(* IEC 61131-3 sources: programs/VI-54/VI-54_20171205/VI-54_20171205/Stations/PLC_VI54/VI-54_171014/Class/SafetyClass, 1 file *)

(* ---- SafetyClass.st ---- *)
(*!
<Class
	Name               = "SafetyClass"
	Revision           = "0.0"
	RealtimeTask       = "false"
	CyclicTask         = "false"
	BackgroundTask     = "false"
	Sigmatek           = "false"
	OSInterface        = "false"
	HighPriority       = "false"
	Automatic          = "false"
	UpdateMode         = "Prescan"
	SharedCommandTable = "true"
	Objectsize         = "(390,300)">
	<Channels>
		<Server Name="SafetyOut1" Visualized="false" Initialize="false" WriteProtected="true" Retentive="false"/>
		<Server Name="SafetyOut2" Visualized="false" Initialize="false" WriteProtected="true" Retentive="false"/>
		<Server Name="SafetyOut3" Visualized="false" Initialize="false" WriteProtected="true" Retentive="false"/>
		<Server Name="SafetyOut4" Visualized="false" Initialize="false" WriteProtected="true" Retentive="false"/>
		<Client Name="CleaningMode" Required="true" Internal="false"/>
		<Client Name="MasterOverrule" Required="true" Internal="false"/>
		<Client Name="SafetyInp1" Required="false" Internal="false"/>
		<Client Name="SafetyInp2" Required="false" Internal="false"/>
		<Client Name="SafetyInp3" Required="false" Internal="false"/>
		<Client Name="SafetyInp4" Required="false" Internal="false"/>
	</Channels>
</Class>
*)
SafetyClass : CLASS
  //Servers:
	SafetyOut1 	: SvrChCmd_DINT;
	SafetyOut2 	: SvrCh_DINT;
	SafetyOut3 	: SvrCh_DINT;
	SafetyOut4 	: SvrCh_DINT;
  //Clients:
	MasterOverrule 	: CltCh_DINT;
	CleaningMode 	: CltCh_DINT;
	SafetyInp1 	: CltCh_DINT;
	SafetyInp2 	: CltCh_DINT;
	SafetyInp3 	: CltCh_DINT;
	SafetyInp4 	: CltCh_DINT;
  //Variables:
  //Functions:

	FUNCTION VIRTUAL GLOBAL SafetyOut1::Read
		VAR_OUTPUT
			output (EAX) 	: DINT;
		END_VAR;

	FUNCTION VIRTUAL GLOBAL SafetyOut2::Read
		VAR_OUTPUT
			output (EAX) 	: DINT;
		END_VAR;

	FUNCTION VIRTUAL GLOBAL SafetyOut3::Read
		VAR_OUTPUT
			output (EAX) 	: DINT;
		END_VAR;

	FUNCTION VIRTUAL GLOBAL SafetyOut4::Read
		VAR_OUTPUT
			output (EAX) 	: DINT;
		END_VAR;
  //Tables:
	FUNCTION @STD
		VAR_OUTPUT
			ret_code	: CONFSTATES;
		END_VAR;
	FUNCTION GLOBAL TAB @CT_;
END_CLASS;

FUNCTION VIRTUAL GLOBAL SafetyClass::SafetyOut1::Read
	VAR_OUTPUT
		output (EAX) 	: DINT;
	END_VAR

  SafetyInp1 := SafetyInp1.Read();
  if MasterOverrule.Read() = 1 | CleaningMode.Read() = 1 then
	  SafetyOut1 := 1;
  else
    SafetyOut1 := SafetyInp1;
  end_if;
  SafetyOut1.Write(input:= SafetyOut1);
  Output := SafetyOut1;

END_FUNCTION

FUNCTION VIRTUAL GLOBAL SafetyClass::SafetyOut2::Read
	VAR_OUTPUT
		output (EAX) 	: DINT;
	END_VAR

  SafetyInp2 := SafetyInp2.Read();
  if MasterOverrule.Read() =  1 | CleaningMode.Read() = 1 then
	  SafetyOut2 := 1;
  else
    SafetyOut2 := SafetyInp2;
  end_if;
  SafetyOut2.Write(input:= SafetyOut2);
  Output := SafetyOut2;

END_FUNCTION

FUNCTION VIRTUAL GLOBAL SafetyClass::SafetyOut3::Read
	VAR_OUTPUT
		output (EAX) 	: DINT;
	END_VAR

  SafetyInp3 := SafetyInp3.Read();
  if MasterOverrule.Read() = 1 | CleaningMode.Read() = 1 then
	  SafetyOut3 := 1;
  else
    SafetyOut3 := SafetyInp3;
  end_if;
  SafetyOut3.Write(input:= SafetyOut3);
  Output := SafetyOut3;

END_FUNCTION

FUNCTION VIRTUAL GLOBAL SafetyClass::SafetyOut4::Read
	VAR_OUTPUT
		output (EAX) 	: DINT;
	END_VAR

  SafetyInp4 := SafetyInp4.Read();
  if MasterOverrule.Read() = 1 | CleaningMode.Read() = 1 then
	  SafetyOut4 := 1;
  else
    SafetyOut4 := SafetyInp4;
  end_if;
  SafetyOut4.Write(input:= SafetyOut4);
  Output := SafetyOut4;

END_FUNCTION
